GLOBALCONSTANTS DefaultPool_Dreieck_Numeric (* Numeric object pool constants (ID, Scale, Offset, Decimals) *)
  PACKAGE Uebungen::const::UT::Dreieck;
  VAR_GLOBAL CONSTANT
    InputNumber_Sollwert_N : logiBUS::utils::conversion::phys::NumericObjectPool_S := (u16ObjId := 9000, r32Scale := 1.0, i32Offset := -42, u8Decimals := 0);
    InputNumber_Istwert_N : logiBUS::utils::conversion::phys::NumericObjectPool_S := (u16ObjId := 9001, r32Scale := 1.0, i32Offset := -42, u8Decimals := 0);
    NumberVariable_Sollwert_N : logiBUS::utils::conversion::phys::NumericObjectPool_S := (u16ObjId := 21000, r32Scale := 1.0, i32Offset := -42, u8Decimals := 0);
    NumberVariable_Istwert_N : logiBUS::utils::conversion::phys::NumericObjectPool_S := (u16ObjId := 21001, r32Scale := 1.0, i32Offset := -42, u8Decimals := 0);
    InputNumber_Messwert_N : logiBUS::utils::conversion::phys::NumericObjectPool_S := (u16ObjId := 9002, r32Scale := 1.0, i32Offset := 0, u8Decimals := 0);
    NumberVariable_Messwert_N : logiBUS::utils::conversion::phys::NumericObjectPool_S := (u16ObjId := 21002, r32Scale := 1.0, i32Offset := 0, u8Decimals := 0);
  END_VAR
END_GLOBALCONSTANTS
